{attribute 'GeneratedUsingTerminal: EL2642-0000-0016'}
{attribute addProperty BoxType "EL2642-0000-0016"}
{attribute addProperty Id "ErrorBOOL1DiagBOOL1Input_cycle_counterBYTE1"}
{attribute addProperty CRC "2238241738"}
{attribute addProperty Size "3"}
TYPE Device_status_8568DBCA :
STRUCT
	{attribute addProperty Name "Error"}
	Error : BOOL;
	{attribute addProperty Name "Diag"}
	Diag : BOOL;
	{attribute addProperty Name "Input_cycle_counter"}
	Input_cycle_counter : BYTE;
END_STRUCT
END_TYPE

(* stored: Version 1.2.0.0, ProductVersion 3.1.4024.11
   DUT Device_status_8568DBCA: Id {adf08a1c-aa0e-46f1-b864-4ce39974b0df} *)
